// TIA Portal project "babu_comparatorsTryOut" (V15)

(* hardware
DEVICE "S7-1200 station_1"  S7-1200 Station
   slot 0: "Rack_0"  S7-1200 Rack  Rack  V1.0
   slot 1: "PLC_1"  CPU 1212C DC/DC/DC  6ES7 212-1AE40-0XB0  V4.2
*)

// ===== PLC "PLC_1"  CPU 1212C DC/DC/DC =====

VAR_GLOBAL   // PLC tag table "Default tag table"
   "INPUT" AT %M0.0 : Bool;
   "POSITIVE SIGNAL" AT %M0.1 : Bool;
   "IN OUT" AT %M0.2 : Bool;
   "OUTPUT" AT %Q0.0 : Bool;
   "IP2" AT %M0.3 : Bool;
   "OP2" AT %Q0.1 : Bool;
   "OP21" AT %Q0.2 : Bool;
   "IP3" AT %M0.4 : Bool;
   "OP3" AT %M0.5 : Bool;
   "OP31" AT %Q0.3 : Bool;
END_VAR

// folder: System blocks/Program resources

DATA_BLOCK "IEC_Counter_0_DB"   // DB1
{ S7_Optimized_Access := 'TRUE' }
AUTHOR : Simatic
FAMILY : IEC
NAME : CNTR
VERSION : 1.0
// stored: InstanceOfName IEC_COUNTER
"IEC_COUNTER"
BEGIN
END_DATA_BLOCK

DATA_BLOCK "IEC_Counter_0_DB_1"   // DB2
{ S7_Optimized_Access := 'TRUE' }
AUTHOR : Simatic
FAMILY : IEC
NAME : CNTR
VERSION : 1.0
// stored: InstanceOfName IEC_COUNTER
"IEC_COUNTER"
BEGIN
END_DATA_BLOCK

// folder: (top level)

ORGANIZATION_BLOCK "Main"   // OB1, LAD, ProgramCycle
TITLE = "Main Program Sweep (Cycle)"
{ S7_Optimized_Access := 'TRUE' }
VERSION : 0.1
   VAR_INPUT
      Initial_Call : Bool;   // Initial call of this OB
      Remanence : Bool;   // =True, if remanent data are available
   END_VAR
   VAR_TEMP   // added for the SCL form of the ladder/FBD networks
      _w1 : Bool;
   END_VAR
BEGIN

REGION Network 1
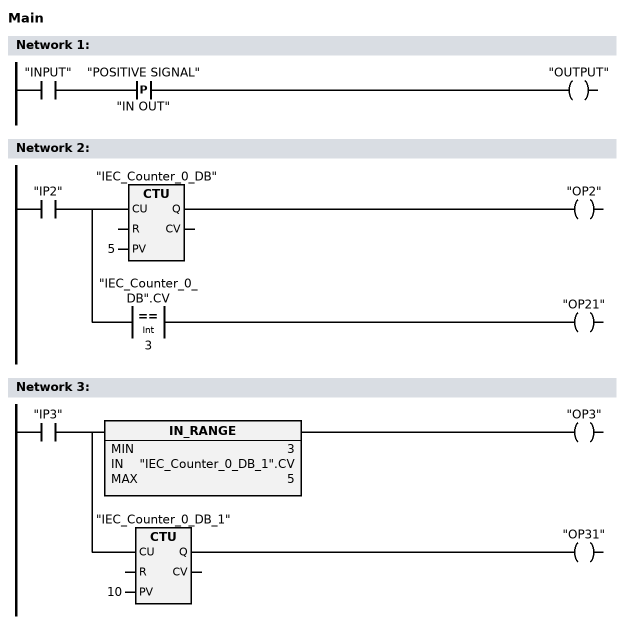
   RUNG wire#powerrail
      Contact( "INPUT" )
      P_Contact(operand := "POSITIVE SIGNAL", bit := "IN OUT")
      Coil( "OUTPUT" )
   END_RUNG
   // the same network as SCL:
   #_w1 := "INPUT" AND "POSITIVE SIGNAL" AND NOT "IN OUT";   // rising edge of "POSITIVE SIGNAL"
   "IN OUT" := "POSITIVE SIGNAL";
   "OUTPUT" := #_w1;
END_REGION

REGION Network 2
   "IEC_Counter_0_DB".CTU(CU := "IP2", PV := 5);
   "OP2" := "IEC_Counter_0_DB".Q;
   "OP21" := "IP2" AND ("IEC_Counter_0_DB".CV = 3);
END_REGION

REGION Network 3
   "OP3" := "IP3" AND (3 <= "IEC_Counter_0_DB_1".CV) AND ("IEC_Counter_0_DB_1".CV <= 5);
   "IEC_Counter_0_DB_1".CTU(CU := "IP3", PV := 10);
   "OP31" := "IEC_Counter_0_DB_1".Q;
END_REGION
END_ORGANIZATION_BLOCK